TYPE ST_DigitalInput_Cfg :
STRUCT
    cfgInvert : BOOL;
END_STRUCT
END_TYPE

(* stored: Version 1.1.0.1, ProductVersion 3.1.4026.12
   DUT ST_DigitalInput_Cfg: Id {b0100001-0001-0000-0000-000000000001} *)
